{attribute 'Tc2GvlVarNames'}
VAR_GLOBAL
END_VAR

(* stored: Version 1.1.0.1, ProductVersion 3.1.4024.0
   GVL Global_Variables: Id {01115cb8-c47a-4ac5-8117-01c0446cddc5} *)
